FUNCTION_BLOCK UdpWindowsSocket IMPLEMENTS ITF_UdpConnection
VAR
	IpAddress			: T_IPv4Addr;
	Port				: UDINT;
	ReceiveBuffer		: ARRAY [0..TCPADS_MAXUDP_BUFFSIZE - 1] OF BYTE;
	
	OpenSocket			: FB_SocketUdpCreate;
	Receive				: FB_SocketUdpReceiveFrom;
	Send				: FB_SocketUdpSendTo;
	SendState			: BYTE;
	Sending 			: BOOL;
	PacketsSent			: ULINT;
	CloseSocket			: FB_SocketClose;
	
	IsConnectionOpen	: BOOL;
END_VAR

METHOD CyclicUpdate : BOOL
VAR
	i	: BYTE;
END_VAR
OpenSocket
(
	sSrvNetId 	:= '', 
	sLocalHost	:= IpAddress, 
	nLocalPort	:= Port, 
);

Send
(
	sSrvNetId	:= '', 
	hSocket		:= OpenSocket.hSocket, 
);

FOR i := 0 TO 9 BY 1 DO
	
	Receive
	(
		sSrvNetId	:= '', 
		hSocket		:= OpenSocket.hSocket, 
		cbLen		:= SIZEOF(ReceiveBuffer), 
		pDest		:= ADR(ReceiveBuffer) 
	);
	
	IF IsSending() OR NOT IsConnectionOpen THEN
	
		Receive(bExecute := FALSE);
		
	ELSE
		
		Receive(bExecute := NOT(Receive.bExecute));
	
	END_IF

END_FOR


CloseSocket
(
	sSrvNetId	:= '', 
	hSocket		:= OpenSocket.hSocket, 
);

IF OpenSocket.hSocket.handle <> 0 AND OpenSocket.bExecute THEN
	
	IsConnectionOpen := TRUE;
	
ELSE

	IsConnectionOpen := FALSE;

END_IF
END_METHOD

//FB_Exit must be implemented explicitly. If there is an implementation, then the
//method is called before the controller removes the code of the function block instance
//(implicit call). The return value is not evaluated.
METHOD FB_Exit: BOOL
VAR_INPUT
    bInCopyCode: BOOL;  // TRUE: the exit method is called in order to leave the instance which will be copied afterwards (online change).  
END_VAR
TryCloseConnection();
END_METHOD

//FB_Init is always available implicitly and it is used primarily for initialization.
//The return value is not evaluated. For a specific influence, you can also declare the
//methods explicitly and provide additional code there with the standard initialization
//code. You can evaluate the return value.
METHOD FB_Init: BOOL
VAR_INPUT
    bInitRetains: BOOL; // TRUE: the retain variables are initialized (reset warm / reset cold)
    bInCopyCode: BOOL;  // TRUE: the instance will be copied to the copy code afterward (online change) 
	IpAddress	: T_IPv4Addr;
	Port		: UDINT;  
END_VAR
THIS^.IpAddress := IpAddress;
THIS^.Port := Port;
END_METHOD

METHOD IsConnected : BOOL
IsConnected := IsConnectionOpen;

RETURN;
END_METHOD

METHOD IsSending : BOOL
IsSending := Sending;

RETURN;
END_METHOD

{warning 'Add property implementation'}
PROPERTY LastReceivedIp : T_IPv4Addr
GET
LastReceivedIp := Receive.sRemoteHost;
END_GET
END_PROPERTY

{warning 'Add property implementation'}
PROPERTY LastReceivedPort : UDINT
GET
LastReceivedPort := Receive.nRemotePort;
END_GET
END_PROPERTY

{warning 'Add property implementation'}
PROPERTY ReceiveBufferReference : REFERENCE TO ARRAY [0..(TCPADS_MAXUDP_BUFFSIZE - 1)] OF BYTE
GET
ReceiveBufferReference REF= ReceiveBuffer;
END_GET
END_PROPERTY

METHOD TryCloseConnection : HRESULT
TryCloseConnection := S_PENDING;

OpenSocket(bExecute := FALSE);

CloseSocket(bExecute := TRUE);

IF OpenSocket.hSocket.handle = 0 THEN
	
	TryCloseConnection := S_OK;

ELSIF OpenSocket.bError THEN

	TryCloseConnection := -1;	

END_IF

RETURN;
END_METHOD

METHOD TryOpenConnection : HRESULT
TryOpenConnection := S_PENDING;

CloseSocket(bExecute := FALSE);

OpenSocket(bExecute := TRUE);

IF OpenSocket.hSocket.handle <> 0 THEN
	
	TryOpenConnection := S_OK;

ELSIF OpenSocket.bError THEN

	TryOpenConnection := -1;	

END_IF

RETURN;
END_METHOD

METHOD TryReadReceiveBuffer : HRESULT
VAR_INPUT
	DataBuffer		: REFERENCE TO ARRAY [0..TCPADS_MAXUDP_BUFFSIZE - 1] OF BYTE;
END_VAR
VAR
	i				: UDINT;
END_VAR
TryReadReceiveBuffer := S_PENDING;

IF ReceiveBuffer[0] = 0 THEN
	
	TryReadReceiveBuffer := -1;

	RETURN;	

END_IF

FOR i := 0 TO TCPADS_MAXUDP_BUFFSIZE BY 1 DO
	
	IF ReceiveBuffer[i] = 0 THEN
		
		EXIT;
		
	END_IF

	DataBuffer[i] := ReceiveBuffer[i];

END_FOR

IF ReceiveBuffer[0] <> 0 THEN
	
	TryReadReceiveBuffer := S_OK;

ELSE

	TryReadReceiveBuffer := -2;

END_IF

RETURN;
END_METHOD

METHOD TrySendData : HRESULT
VAR_INPUT
	IpAddress		: T_IPv4Addr;
	Port			: UDINT;
	DataAddress		: PVOID;
	DataLength		: UDINT;
END_VAR
TrySendData := S_PENDING;

IF NOT IsConnected() THEN
	
	TrySendData := -1;
	
	RETURN;

END_IF

Send
(
	sRemoteHost	:= IpAddress, 
	nRemotePort	:= Port, 
	cbLen		:= DataLength, 
	pSrc		:= DataAddress, 
	bExecute	:= TRUE, 
);

Sending := TRUE;

CASE SendState OF
	
	0:
	
		IF Send.bBusy THEN
			
			SendState := 1;
			
		END_IF



	1:
	
		IF Send.bError THEN
			
			Send(bExecute := FALSE);
			
			TrySendData := -1;
			
			SendState := 0;
			
			Sending := FALSE;
			
			RETURN;
		
		ELSIF NOT Send.bBusy THEN
			
			Send(bExecute := FALSE);
		
			TrySendData := S_OK;
			
			PacketsSent := PacketsSent + 1;
			
			SendState := 0;
			
			Sending := FALSE;
			
			RETURN;
		
		END_IF
END_CASE
END_METHOD

END_FUNCTION_BLOCK

(* stored: Version 1.1.0.1
   POU UdpWindowsSocket: Id {ad35c0b7-db8d-4688-9112-1457484c5200}, SpecialFunc None
   Folder ITF_UdpConnection: Id {6e849f84-8864-4f97-8eeb-b3d2c78f1ae2}
   Method CyclicUpdate: Id {b6d2a984-cd64-4493-bdc6-c52c97bcd1ff}
   Method FB_Exit: Id {09fa55a5-0e45-4172-ae61-55feadab3ce8}
   Method FB_Init: Id {15efff28-c652-4b7e-9b7c-7c0e8ce42ddc}
   Method IsConnected: Id {8f4c16ee-1759-41ca-9d3c-5334496d7d18}
   Method IsSending: Id {13e6fe11-2ce9-4072-a618-52bebb948349}
   Property LastReceivedIp: Id {1be0fcdb-6c80-41d0-8463-11d58649fa80}
   Get Get: Id {9284e367-4412-4008-b229-2bd469f707d3}
   Property LastReceivedPort: Id {a3bba1ac-ec01-40a6-b89d-1cf870cb9c74}
   Get Get: Id {8db3583f-bc06-41ef-b2ad-28b4e5aca0c5}
   Property ReceiveBufferReference: Id {f4d6b744-2f99-48da-b241-cf7eb4cefdcd}
   Get Get: Id {a0b1ba46-ae51-4579-baf6-f1a850ff7a54}
   Method TryCloseConnection: Id {752fc699-79a0-4dfb-92d8-5930e09a3363}
   Method TryOpenConnection: Id {638b00cb-58aa-4579-8647-331293c7c671}
   Method TryReadReceiveBuffer: Id {93010522-48e9-47c9-83a5-b0a64bd21a0c}
   Method TrySendData: Id {910c1629-032b-4b69-b3a6-02b4be236a07} *)
